(* PLC project CDPR_4cables, Beckhoff Automation GmbH TwinCAT PLC Control 3.5.13.21 *)
(* stored: creationDateTime 2024-03-19T20:38:32.9552202, modificationDateTime 2024-03-19T20:38:32.9572148 *)

PROGRAM MAIN
VAR
	invKin_solution: ARRAY [1..4] OF REAL;//solution for the backward kinematics
	dirKinSph_solution: Pose3D;				//solution for the forward kinematics spheres' method
	dirKinNR_solution: Pose3D;				//solution for the forward kinematics newton-raphson
	pObj: Pose3D := (x := -100, y := 175, z := 500);
	l: ARRAY [1..4] OF REAL := [1362.06030, 1421.83276, 1223.78845, 1153.80164];
	q: ARRAY [1..4] OF Pose3D;
	m: ARRAY [1..4] OF Pose3D;
	pIni: Pose3D;
	threshold: REAL:=0.01;
	wp: WorkspaceLimits := (LimitX_neg := -500, LimitX_pos := 500, LimitY_neg := -800, LimitY_pos := 800, LimitZ_neg := 0, LimitZ_pos := 1600);
END_VAR

            q:=GetQvectors(58.0,0,103.0);
m:=GetMvectors(890.0,1450.0,1520);
invKin_solution:=InvKin_4cables(q:=q,m:=m,pObj:=pObj);
dirKinSph_solution:=DirKin_4cables_Sphere(q:=q,m:=m,l:=l,wp:=wp);
dirKinNR_solution:=DirKin_4cables_NR(q:=q,m:=m,l:=l,pIni:=pIni,threshold:=threshold,iterations:=100);
          
END_PROGRAM
